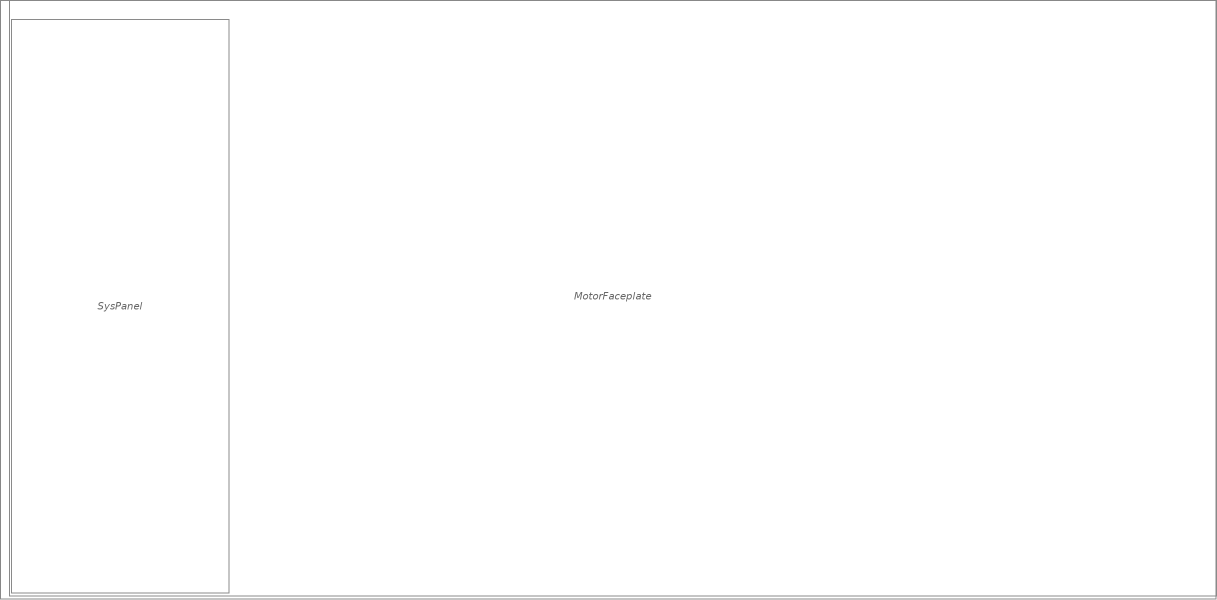
VISUALIZATION Main  // 1217x600
    TabControl (9,-4 1208x600)
        shows MotorFaceplate()
        shows MotorFaceplate2()
        [0]: TabTitle=Drive 1: Manual Control
        [1]: TabTitle=Drive 2
    Frame (11,19 218x574)
        shows SysPanel()
END_VISUALIZATION

(* stored: Version 1.1.0.1, ProductVersion 3.1.4024.12
   Visu Main: Id {5e223294-ed9a-4657-8444-2386fbb117d8} *)
